# B&R Automation Studio project prac3
Automation Studio 4.5.2.102

## Configuration Config1

CPU 4PP065.0571-P74, AutomationRuntime D4.52, Build 4.1.2, Vc V4.52.0, Safety 1.10

### Task classes (Cpu.sw)
```
Cyclic#1:
  Program <- Program.prg
DataObjects: Acp10sys
NcDataObjects: acp10etxen <- acp10etxen.dob
VcDataObjects: Visu <- Visu.dob
Binaries: udbdef, TCData, Role, sysconf, ashwd, ashwac, asfw, iomap, User, arconfig, Acp10map, acp10cfg
Libraries: Acp10man, Acp10par, NcGlobal, Acp10sdc, AsBrStr, sys_lib, runtime, Library, powerlnk, astime, fileio
```

### Hardware
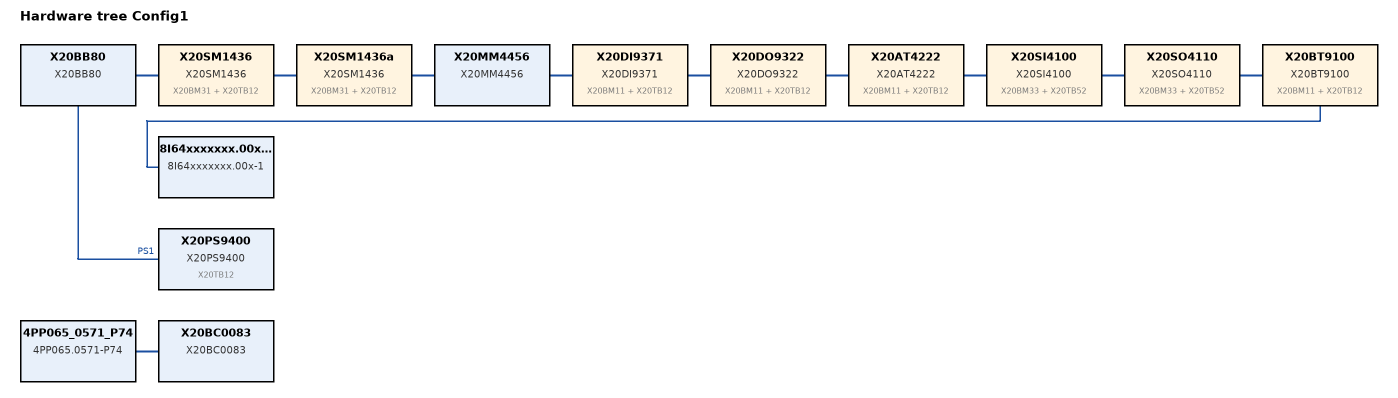
```
4PP065_0571_P74 : 4PP065.0571-P74 v1.1.2.0
  Connector IF5:
    ActivateDevice = 1
    Mode = Manual
    InternetAddress = 10.0.1.10
    SubnetMask = 255.255.255.0
  ConfigurationID = labBR
  TimerDeviceType = EPLX2X
  TimerDevice = 4PP065_0571_P74.IF4
  TaskClassIdleTime = 2000
  Cyclic1Output = 1
  VcObjectName = Visu
8I64xxxxxxx.00x-1 : 8I64xxxxxxx.00x-1 v2.1.3.0  [X2X1 -> X20BT9100.X2X1 [Cable Type=X2XCable, Length=10, Version=1.0.0.2]]
  FunctionModel = Standard
  packedETAD = packed
  packedCMDD = packed
X20AT4222 : X20AT4222 v1.2.3.0  [SS1 -> X20TB12e.SS; SL -> X20BM11b.SL1]
X20BB80 : X20BB80 v1.0.2.0
X20BC0083 : X20BC0083 v2.9.0.0  [PLK1 -> 4PP065_0571_P74.IF4 (NodeNumber=2) [Cable Type=PowerlinkCable, Length=10, Version=1.0.0.2]; SL -> X20BB80.SL1]
X20BM11 : X20BM11 v1.0.0.1  [X2X1 -> X20MM4456.X2X2]
X20BM11a : X20BM11 v1.0.0.1  [X2X1 -> X20BM11.X2X2]
X20BM11b : X20BM11 v1.0.0.1  [X2X1 -> X20BM11a.X2X2]
X20BM11c : X20BM11 v1.0.0.1  [X2X1 -> X20BM33a.X2X2]
X20BM31 : X20BM31 v1.0.0.1  [X2X1 -> X20BB80.IF1]
X20BM31a : X20BM31 v1.0.0.1  [X2X1 -> X20BM31.X2X2]
X20BM33 : X20BM33 v1.0.0.4  [X2X1 -> X20BM11b.X2X2]
X20BM33a : X20BM33 v1.0.0.4  [X2X1 -> X20BM33.X2X2]
X20BT9100 : X20BT9100 v1.0.3.0  [SS1 -> X20TB12f.SS; SL -> X20BM11c.SL1]
X20DI9371 : X20DI9371 v1.0.2.0  [SS1 -> X20TB12c.SS; SL -> X20BM11.SL1]
X20DO9322 : X20DO9322 v1.0.3.0  [SS1 -> X20TB12d.SS; SL -> X20BM11a.SL1]
X20MM4456 : X20MM4456 v1.1.5.0  [X2X1 -> X20BM31a.X2X2]
X20PS9400 : X20PS9400 v1.8.0.0  [SS1 -> X20TB12.SS; PS -> X20BB80.PS1]
X20SI4100 : X20SI4100 v1.10.1.1  [SS1 -> X20TB52a.SS; SL -> X20BM33.SL1]
X20SM1436 : X20SM1436 v1.4.2.1  [SS1 -> X20TB12a.SS; SL -> X20BM31.SL1]
X20SM1436a : X20SM1436 v1.4.2.1  [SS1 -> X20TB12b.SS; SL -> X20BM31a.SL1]
X20SO4110 : X20SO4110 v1.10.1.1  [SS1 -> X20TB52b.SS; SL -> X20BM33a.SL1]
  SafeModuleID = 3
X20TB12 : X20TB12 v1.0.0.0
X20TB12a : X20TB12 v1.0.0.0
X20TB12b : X20TB12 v1.0.0.0
X20TB12c : X20TB12 v1.0.0.0
X20TB12d : X20TB12 v1.0.0.0
X20TB12e : X20TB12 v1.0.0.0
X20TB12f : X20TB12 v1.0.0.0
X20TB52a : X20TB52 v1.0.0.1
X20TB52b : X20TB52 v1.0.0.1
```

### IoMap.iom - 4PP065_0571_P74/IoMap.iom
```iecst
VAR_CONFIG
	::Program:EVIRD.STATE AT %IW."8I64xxxxxxx.00x-1".ETAD_Input;
	::Program:EVIRD.COMMAND AT %QW."8I64xxxxxxx.00x-1".CMDD_Output;
	::Program:speed AT %QW."8I64xxxxxxx.00x-1".LFRD_Output;
	::Program:EVIRD.TORQUE AT %IW."8I64xxxxxxx.00x-1".OTR_Input;
END_VAR
```

## Logical view

### Library Logical/Library (ANSIC)

#### Constants.var
```iecst
VAR CONSTANT
	STATE_DISABLED : USINT := 64;
	STATE_SWITCHED_ON : USINT := 35;
	STATE_READY : USINT := 33;
	CMD_SWITCHED_ON : USINT := 7;
	CMD_ENABLED : USINT := 15;
	CMD_SHUTDOWN : USINT := 6;
END_VAR
```

#### Library.fun
```iecst
{REDUND_ERROR} FUNCTION_BLOCK DRIVE (*TODO: Add your comment here*) (*$GROUP=User,$CAT=User,$GROUPICON=User.png,$CATICON=User.png*)
	VAR_INPUT
		STATE : UINT;
		ENABLE : BOOL;
	END_VAR
	VAR_OUTPUT
		COMMAND : UINT;
	END_VAR
	VAR_INPUT
		TORQUE : INT;
	END_VAR
END_FUNCTION_BLOCK
```

#### DRIVE.c
```c
#include <bur/plctypes.h>
#ifdef __cplusplus
	extern "C"
	{
#endif
	#include "Library.h"
#ifdef __cplusplus
	};
#endif
/* TODO: Add your comment here */
void DRIVE(struct DRIVE* inst)
{
	UINT mask = inst->STATE & 0x6f;
	if (!inst->ENABLE)
	{
		inst->COMMAND=CMD_SHUTDOWN;
	}
	else
	{
		switch(mask)
		{
			case STATE_DISABLED:

				inst->COMMAND=CMD_SHUTDOWN;
				break;

			case STATE_READY:

				inst->COMMAND=CMD_ENABLED;
				break;

			case STATE_SWITCHED_ON:

				inst->COMMAND=CMD_SWITCHED_ON;
				break;

		}
	}
	/*TODO: Add your code here*/
}
```

### Program Logical/Program (ANSIC)

#### Variables.var
```iecst
VAR
	speed : INT;
	EVIRD : DRIVE;
	speedPlus : BOOL;
	speedMinus : BOOL;
	reset : BOOL;
	reverse : BOOL;
END_VAR
```

#### Main.c
```c
#include <bur/plctypes.h>

#ifdef _DEFAULT_INCLUDES
	#include <AsDefault.h>
#endif

void _INIT ProgramInit(void)
{
	speed = 1000;
	EVIRD.ENABLE=1;
}

void _CYCLIC ProgramCyclic(void)
{
	DRIVE(&EVIRD);
	if ( speedPlus == 1 )
	{
		speed +=1;
	}
	if ( speedMinus == 1 )
	{
		speed -=1;
	}
	if (reverse == 1)
	{
		speed = -speed;
	}
	if(reset == 1)
	{
		speed = 1000;
		EVIRD.ENABLE=1;
	}
	if (speed>=2000)
	{
		speed = 2000;
	}
	if (speed<= -2000)
	{
		speed = -2000;
	}
}

void _EXIT ProgramExit(void)
{

}
```

- Visualisation Logical/Visu (not shown)

Listed in the project but not available here: Logical/Global.typ, Logical/Global.var, Logical/Libraries, Logical/acp10etxen
